// TIA Portal V19 export
FUNCTION "FC_Pos_Manager" : Void   // FC50, STL
TITLE = Positionsmanager
{ S7_Optimized_Access := 'FALSE' }
// Bearbeitung und Aktualisierung der Positionen
// in jedem Zyklus wird eine im DB1 definierte Anzahl von Positionen bearbeitet.
// stored: AutoNumber false
   VAR_TEMP
      count : Int;   // Zähler Pos pro Zyklus
      akt_Pos : USInt;   // aktuelle Position
      DummyPos : Bool;   // Position nicht behandeln
   END_VAR
BEGIN

NETWORK
TITLE = Umlauf Pos per Zyklus
// Umlaufzähler verwalten für Positionsbearbeitung
//----------------------------------
//Umlauf
//----------------------------------
      L     "DB_ANLAGE".config.ANZ_POS_per_Cyc;
schl: T     #count;

      L     "DB_POS".akt_POS;
      L     1;
      <I;
      JC    nok;
      L     "DB_POS".akt_POS;
      L     "DB_ANLAGE".config.ANZ_Pos;
      <=I;
      JC    go;

nok:  L     1;
      T     "DB_POS".akt_POS;

go:   L     "DB_POS".akt_POS;
      T     #akt_Pos;
//---------------------------------
//laden der Positionsdaten
//---------------------------------
      CALL  "FC_POS_TO_WORK"
      ( Akt_Pos  := #akt_Pos,
        not_load := #DummyPos
      );

//----------------------------------
//Position geladen --> Behandlung
//----------------------------------
      A     #DummyPos;
      JC    nexP;


NETWORK
TITLE = Badbehandlung
// Bearbeitung der Positionen und Aktualisierung von PC-Daten

      CALL  "FC_Pos_Behandlung"
      ( Pos_Nr     := #akt_Pos,
        send_DBEvt := TRUE
      );


NETWORK
TITLE = Rückladen der Positionsdaten
// Daten werden aus dem Arbeitsbereich wieder ausgelagert
//----------------------------------
//zurück laden der Positionsdaten
//----------------------------------
      CALL  "FC_WORK_TO_POS"
      ( Akt_Pos := #akt_Pos
      );
//----------------------------------
//Zeiger auf nächste Position setzen
//----------------------------------
nexP: L     "DB_POS".akt_POS;
      L     1;
      +I;
      T     "DB_POS".akt_POS;
//----------------------------------
//Zählschleifenrücksprung
//----------------------------------
      L     #count;
      LOOP  schl;
      BE;
END_FUNCTION
